TEXTLIST ExtendedFadeTime
  0 = 'No Fade'
  1 = '1 * 100 ms = 100 ms'
  2 = '2 * 100 ms = 200 ms'
  3 = '3 * 100 ms = 300 ms'
  4 = '4 * 100 ms = 400 ms'
  5 = '5 * 100 ms = 500 ms'
  6 = '6 * 100 ms = 600 ms'
  7 = '7 * 100 ms = 700 ms'
  8 = '8 * 100 ms = 800 ms'
  9 = '9 * 100 ms = 900 ms'
  10 = '10 * 100 ms = 1000 ms'
  11 = '11 * 100 ms = 1100 ms'
  12 = '12 * 100 ms = 1200 ms'
  13 = '13 * 100 ms = 1300 ms'
  14 = '14 * 100 ms = 1400 ms'
  15 = '15 * 100 ms = 1500 ms'
  16 = '16 * 100 ms = 1600 ms'
  17 = '1 * 1 s = 1 s'
  18 = '2 * 1 s = 2 s'
  19 = '3 * 1 s = 3 s'
  20 = '4 * 1 s = 4 s'
  21 = '5 * 1 s = 5 s'
  22 = '6 * 1 s = 6 s'
  23 = '7 * 1 s = 7 s'
  24 = '8 * 1 s = 8 s'
  25 = '9 * 1 s = 9 s'
  26 = '10 * 1 s = 10 s'
  27 = '11 * 1 s = 11 s'
  28 = '12 * 1 s = 12 s'
  29 = '13 * 1 s = 13 s'
  30 = '14 * 1 s = 14 s'
  31 = '15 * 1 s = 15 s'
  32 = '16 * 1 s = 16 s'
  33 = '1 * 10 s = 10 s'
  34 = '2 * 10 s = 20 s'
  35 = '3 * 10 s = 30 s'
  36 = '4 * 10 s = 40 s'
  37 = '5 * 10 s = 50 s'
  38 = '6 * 10 s = 60 s'
  39 = '7 * 10 s = 70 s'
  40 = '8 * 10 s = 80 s'
  41 = '9 * 10 s = 90 s'
  42 = '10 * 10 s = 100 s'
  43 = '11 * 10 s = 110 s'
  44 = '12 * 10 s = 120 s'
  45 = '13 * 10 s = 130 s'
  46 = '14 * 10 s = 140 s'
  47 = '15 * 10 s = 150 s'
  48 = '16 * 10 s = 160 s'
  49 = '1 * 1 min = 1 min'
  50 = '2 * 1 min = 2 min'
  51 = '3 * 1 min = 3 min'
  52 = '4 * 1 min = 4 min'
  53 = '5 * 1 min = 5 min'
  54 = '6 * 1 min = 6 min'
  55 = '7 * 1 min = 7 min'
  56 = '8 * 1 min = 8 min'
  57 = '9 * 1 min = 9 min'
  58 = '10 * 1 min = 10 min'
  59 = '11 * 1 min = 11 min'
  60 = '12 * 1 min = 12 min'
  61 = '13 * 1 min = 13 min'
  62 = '14 * 1 min = 14 min'
  63 = '15 * 1 min = 15 min'
  64 = '16 * 1 min = 16 min'
  255 = 'Unknown'
   = ''
END_TEXTLIST

(* stored: Version 1.1.0.1
   TextList ExtendedFadeTime: Id {517275cb-6031-487b-9d2e-3a4dddf36bd6} *)
